Yaskawa INFORM job: SQUARE5.JBI

/JOB
//NAME SQUARE5
//POS
///NPOS 5,0,0,0,0,0
///TOOL 0
///POSTYPE PULSE
///PULSE
C00000=-3626,25307,0,0,-64000,-407
C00001=-2626,25307,0,0,-64000,-407
C00002=-2626,26307,0,0,-64000,-407
C00003=-3626,26307,0,0,-64000,-407
C00004=-3626,25307,0,0,-64000,-407
//INST
///DATE 2026/01/21 16:46
///ATTR SC,RW
///GROUP1 RB1
NOP
MOVJ C00000 VJ=25.00
MOVL C00001 V=375.0
MOVJ C00002 VJ=25.00
MOVL C00003 V=375.0
MOVJ C00004 VJ=25.00
END
